INTERFACE I_AsynchronousRpcHandlers

PROPERTY PUBLIC HasHandlers : BOOL
GET
END_GET
END_PROPERTY

METHOD PUBLIC RegisterHandler
VAR_INPUT
	MethodName : T_MAXSTRING;
	Handler : I_AsynchronousRpcHandler;
END_VAR
END_METHOD

METHOD PUBLIC TryGetByMethodName : BOOL
VAR_INPUT
	MethodName : T_MAXSTRING;
	Destination : REFERENCE TO I_AsynchronousRpcHandler;
END_VAR
END_METHOD

END_INTERFACE

(* stored: Version 1.1.0.1, ProductVersion 3.1.4024.12
   Itf I_AsynchronousRpcHandlers: Id {13940dd9-7f39-4e5e-a811-91d182fce911}
   Property HasHandlers: Id {bd9387be-4796-42a8-8f8f-c10df9a654ad}
   Get Get: Id {02f767ed-5ff3-4e8a-9b16-2da38e569d19}
   Method RegisterHandler: Id {0de87ed5-a768-44ec-8b6c-e64dad203ee5}
   Method TryGetByMethodName: Id {d8a72e36-8391-4809-a02c-6c3752183eca} *)
